PROGRAM RobotDynamics

VAR
	// slave robot arms joint data
	m_slaveJointsData AT %I* :ST_SlaveJointData;
	
	// setup joint5 position
	m_setupJointData AT %I* :ST_SetupJointData;
	
	// instrument info
	m_instruInfo AT %I* :ARRAY[1..g_sArmNum] OF ST_InstruStatus;
	
	// dynamic output
	m_slaveDynaData AT %Q* : ST_SlaveDynaData;
	m_setupJnt3Gravity AT %Q* : LREAL;
	m_setupJnt5Gravity AT %Q* : LREAL;
	
	// flag to init robot dynamic model
	m_robotDynaInit :BOOL :=FALSE;
	
	// grivity model block
	m_gravityModel :ARRAY[1..g_sArmNum] OF FB_SlaveGravity;
	m_gravityModelFull :ARRAY[1..g_sArmNum] OF FB_SetupSlaveGravity;
	

	// code execute time measure
	m_codeTime : Profiler;
	
	i: INT;
	
END_VAR

m_codeTime(START:=TRUE, RESET:=TRUE);

// robot dynamic model init
IF m_robotDynaInit =FALSE THEN
	FOR i:=1 TO g_sArmNum DO
		m_gravityModel[i].Init(i);
	END_FOR

	m_robotDynaInit:=TRUE;
END_IF

// run gravity model
FOR i:=1 TO g_sArmNum DO
	m_slaveDynaData.m_gravity[i]:=m_gravityModel[i].run(m_setupJointData.m_curJntPos[i][5], m_slaveJointsData.m_curJntPos[i],m_instruInfo[i]);
//	m_gravityModelFull[i].run(m_setupJointData.m_curJntPos[i], m_slaveJointsData.m_curJntPos[i],m_instruInfo[i],
//				o_setupJ3Gravity=>m_setupJnt3Gravity, o_setupJ5Gravity=>m_setupJnt5Gravity, o_slaveGravity=>m_slaveDynaData.m_gravity);
END_FOR

m_codeTime(START:=FALSE);

END_PROGRAM

(* stored: Version 1.1.0.1, ProductVersion 3.1.4024.12
   POU RobotDynamics: Id {798b314f-0a53-4e08-997d-5fefed426c86}, SpecialFunc None *)
